{attribute 'linkalways'} 
{attribute 'no_explicit_call' := 'This FB is a CLASS and must be accessed using methods or properties'}
{attribute 'enable_dynamic_creation'}
FUNCTION_BLOCK Node_F_VN_MinElementElementwise_REAL EXTENDS VisionNode
VAR
    ipContainer : _ITcVnContainer;
    fMin : _REAL(0.0);
    hrPrev : _HRESULT(S_OK);
    hresult : _HRESULT(S_OK);
END_VAR

METHOD PUBLIC  Clone : I_Node
VAR
	pNode : POINTER TO Node_F_VN_MinElementElementwise_REAL;
END_VAR
pNode := __NEW(Node_F_VN_MinElementElementwise_REAL);
Clone := pNode^;
END_METHOD

METHOD FB_init : BOOL
VAR_INPUT
	bInitRetains : BOOL; // if TRUE, the retain variables are initialized (warm start / cold start)
	bInCopyCode : BOOL;  // if TRUE, the instance afterwards gets moved into the copy code (online change)
END_VAR
AddInput('ipContainer', ipContainer);
AddInput('hrPrev', hrPrev);
AddOutput('ipContainer', ipContainer);
AddOutput('fMin', fMin);
AddOutput('hresult',hresult);
END_METHOD

METHOD PROTECTED OnExecute
hresult.Value := F_VN_MinElementElementwise_REAL(
    ipContainer := ipContainer.Value,
    fMin := fMin.Value,
    hrPrev:= hrPrev.Value);
END_METHOD

METHOD PUBLIC PreExecutionCheck
VAR_INPUT
	Check : I_PreExecutionChecks;
END_VAR
Check.IsTrue(ipContainer.IsValid, 'ipContainer must be a valid container');
Check.IsTrue(ipContainer.IsType(TC_GLOBAL_CONST_LIST.ContainerType_Vector_REAL), 'ipContainer contains incorrect type');
END_METHOD

END_FUNCTION_BLOCK

(* stored: Version 1.1.0.1, ProductVersion 3.1.4026.13
   POU Node_F_VN_MinElementElementwise_REAL: Id {bf9ce613-8ec7-418a-beaf-24dcbe34fdd9}, SpecialFunc None
   Folder Constructor: Id {eed0ff0e-3792-4e0b-988a-a0ecf4d5cf51}
   Method Clone: Id {bb48f35e-48aa-49c4-80c8-bbe06fc3f5c9}
   Method FB_init: Id {fa4d0908-ebf9-4ccb-aec7-95a8fd196a87}
   Method OnExecute: Id {e4329ea6-7687-4dd8-9338-5b6f03a54144}
   Method PreExecutionCheck: Id {b4462643-2b7e-45bf-a9a4-5cafbe8e8e45} *)
